
TYPE "_AV LILESH_SND"
VERSION : 0.1
   STRUCT
      LILESH_ID { ExternalAccessible := 'False'; ExternalVisible := 'False'; ExternalWritable := 'False';  WaveWritable := 'False'} : Byte;   //  ROS->AV 1=ROS; 2 =Crane; 3 = Block ||AV->ROS 4 = AV ||5= Crane AV F; 6=Yard AV Fault
      WATCHDOG_LILESH { ExternalAccessible := 'False'; ExternalVisible := 'False'; ExternalWritable := 'False';  WaveWritable := 'False'} : Byte;   // Running watchdog number
      FIRST_INDEX { ExternalAccessible := 'False'; ExternalVisible := 'False'; ExternalWritable := 'False';  WaveWritable := 'False'} : Byte;   // 1…N
      LAST_INDEX { ExternalAccessible := 'False'; ExternalVisible := 'False'; ExternalWritable := 'False';  WaveWritable := 'False'} : Byte;   // 1…N
      lilesh_1 { ExternalAccessible := 'False'; ExternalVisible := 'False'; ExternalWritable := 'False';  WaveWritable := 'False'} : Byte;
      lilesh_2 { ExternalAccessible := 'False'; ExternalVisible := 'False'; ExternalWritable := 'False';  WaveWritable := 'False'} : Byte;
      lilesh_3 { ExternalAccessible := 'False'; ExternalVisible := 'False'; ExternalWritable := 'False';  WaveWritable := 'False'} : Int;
      lilesh_4 { ExternalAccessible := 'False'; ExternalVisible := 'False'; ExternalWritable := 'False';  WaveWritable := 'False'} : Int;
   END_STRUCT;

END_TYPE

DATA_BLOCK "A/V312 CPLC  --> A/V CRANE DATA"
TITLE = Crane information to AV
{ DB_Accessible_From_OPC_UA := 'FALSE' ;
 S7_Optimized_Access := 'FALSE' }
VERSION : 2.2
   STRUCT
      LILESH : Array[1..10] of  "_AV LILESH_SND";
   END_STRUCT;


BEGIN

END_DATA_BLOCK

